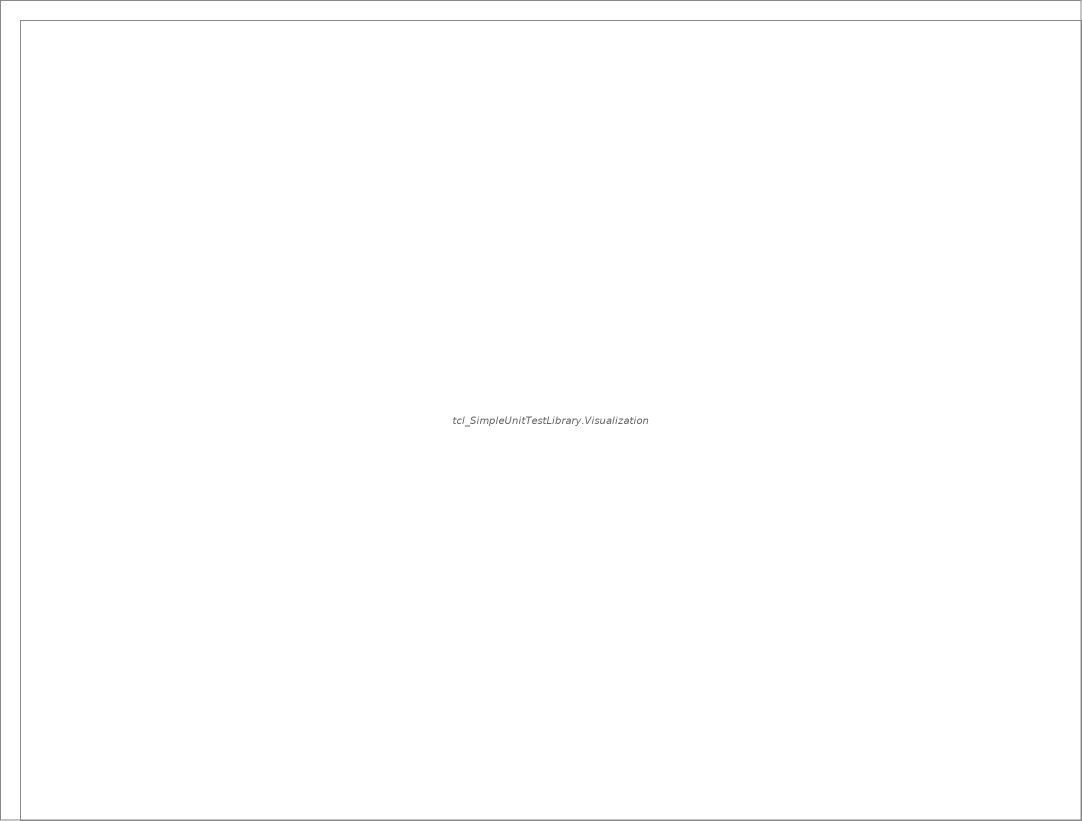
VISUALIZATION Visualization  // 1082x821
    Frame (20,20 1062x801)
        shows tcl_SimpleUnitTestLibrary.Visualization(TestRunner := PB_TestRunner.TestRunner, AssertionMessages := PB_TestRunner.TestRunner.AssertionMessages)
END_VISUALIZATION

(* stored: Version 1.1.0.1, ProductVersion 3.1.4024.6
   Visu Visualization: Id {f7630f05-a200-0986-2471-7edcb76a9027} *)
